{attribute 'qualified_only'}
{attribute 'strict'}
TYPE E_Step :
(
	// special steps
	NoStep := -32767,	// nessuno step
	Unknown := -32000,	// step sconosciuto
	
	// Not Enabled or Errors
	NeOrError := -990,	// SE, non abilitata o in errore
	
	// Recovery
	Recovering := 990,	// SA, ripristino dopo errore

	// Stopping
	Stopping := 900,	// Fase di spegnimento nominale
	
	// Stop
	Stop := 0, 			// S0, stop
	
	// working steps
	Waiting	:= 100,		// S1, attesa oggetto
	Feeding := 200,		// S2, trasferimento oggetto
	Unloading := 300	// S3, scarico oggetto in uscita 
   
);
END_TYPE
//  NoStep = '-32767'
//  Unknown = '-32000'
//  NeOrError = '-990'

(* stored: Version 1.1.0.1, ProductVersion 3.1.4024.12
   EnumerationTextList E_Step: Id {55de7b00-de84-4f53-a951-c988b78497f3} *)
